{attribute 'linkalways'} 
{attribute 'no_explicit_call' := 'This FB is a CLASS and must be accessed using methods or properties'}
{attribute 'enable_dynamic_creation'}
FUNCTION_BLOCK FINAL EQ_UDINT EXTENDS Node
VAR
	in1 : _UDINT(0);
	in2 : _UDINT(0);
	out : _BOOL(FALSE);
END_VAR

METHOD PUBLIC Clone : I_Node
VAR
	pNode : POINTER TO EQ_UDINT;
END_VAR
pNode := __NEW(EQ_UDINT);
Clone := pNode^;
END_METHOD

METHOD FB_init : BOOL
VAR_INPUT
	bInitRetains : BOOL; // if TRUE, the retain variables are initialized (warm start / cold start)
	bInCopyCode : BOOL;  // if TRUE, the instance afterwards gets moved into the copy code (online change)
END_VAR
AddInput('in1',THIS^.in1);
AddInput('in2',THIS^.in2);
AddOutput('out', THIS^.out);
END_METHOD

METHOD PROTECTED OnExecute
VAR
END_VAR
out.Value := in1.Value = in2.Value;
END_METHOD

END_FUNCTION_BLOCK

(* stored: Version 1.1.0.1, ProductVersion 3.1.4024.15
   POU EQ_UDINT: Id {8a19852d-1f40-449c-8727-a46cf7ec3872}, SpecialFunc None
   Folder Constructor: Id {bd5bfc8c-1659-4258-a781-323a81bd9b85}
   Method Clone: Id {f84758f9-789d-4373-bbb8-5d7f0d48767d}
   Method FB_init: Id {051ffc12-61cb-4980-957d-ad9c12b74e1a}
   Method OnExecute: Id {fb5ef3dc-6428-46af-b247-a7c202141af6} *)
